Yaskawa INFORM job: CHECKTOOL4-LONG-45.JBI

/JOB
//NAME CHECKTOOL4-LONG-45
///FOLDERNAME TCP-CHECK-POINT
//POS
///NPOS 4,0,0,0,0,0
///TOOL 4
///POSTYPE PULSE
///PULSE
C00000=0,-80000,-25000,0,-113945,0
C00001=76615,-63731,-18371,0,-109664,-25974
C00002=77854,-64228,-92943,-37751,-90742,58883
C00003=113155,-93155,-94784,1,-77761,-38362
//INST
///DATE 2021/10/07 09:22
///ATTR SC,RW
///GROUP1 RB1
NOP
MOVJ C00000 VJ=50.00
MOVJ C00001 VJ=50.00
MOVL C00002 V=750.0
MOVL C00003 V=750.0
GETS PX040 $PX001
END
